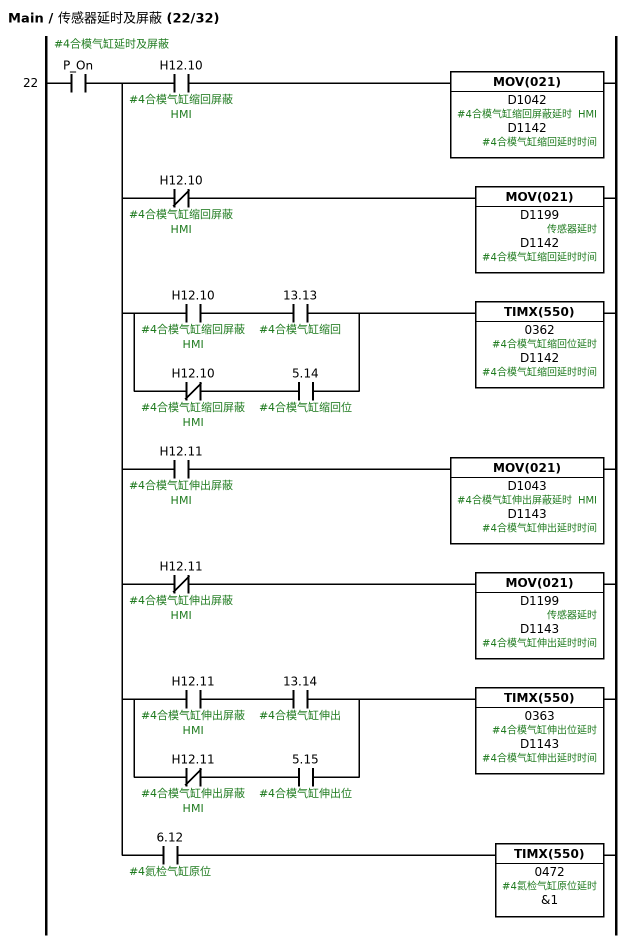
; [picture p24: Main / 传感器延时及屏蔽, rungs 22-22]
; rung 22: #4合模气缸延时及屏蔽
LD P_On
OUT TR0
AND H12.10  ; #4合模气缸缩回屏蔽  HMI
MOV(021) D1042 D1142  ; #4合模气缸缩回屏蔽延时  HMI, #4合模气缸缩回延时时间
LD TR0
ANDNOT H12.10  ; #4合模气缸缩回屏蔽  HMI
MOV(021) D1199 D1142  ; 传感器延时, #4合模气缸缩回延时时间
LD TR0
LD H12.10  ; #4合模气缸缩回屏蔽  HMI
AND 13.13  ; #4合模气缸缩回
LDNOT H12.10  ; #4合模气缸缩回屏蔽  HMI
AND 5.14  ; #4合模气缸缩回位
ORLD
ANDLD
TIMX(550) 0362 D1142  ; #4合模气缸缩回延时时间, #4合模气缸缩回位延时
LD TR0
AND H12.11  ; #4合模气缸伸出屏蔽  HMI
MOV(021) D1043 D1143  ; #4合模气缸伸出屏蔽延时  HMI, #4合模气缸伸出延时时间
LD TR0
ANDNOT H12.11  ; #4合模气缸伸出屏蔽  HMI
MOV(021) D1199 D1143  ; 传感器延时, #4合模气缸伸出延时时间
LD TR0
LD H12.11  ; #4合模气缸伸出屏蔽  HMI
AND 13.14  ; #4合模气缸伸出
LDNOT H12.11  ; #4合模气缸伸出屏蔽  HMI
AND 5.15  ; #4合模气缸伸出位
ORLD
ANDLD
TIMX(550) 0363 D1143  ; #4合模气缸伸出延时时间, #4合模气缸伸出位延时
LD TR0
AND 6.12  ; #4氦检气缸原位
TIMX(550) 0472 &1  ; #4氦检气缸原位延时

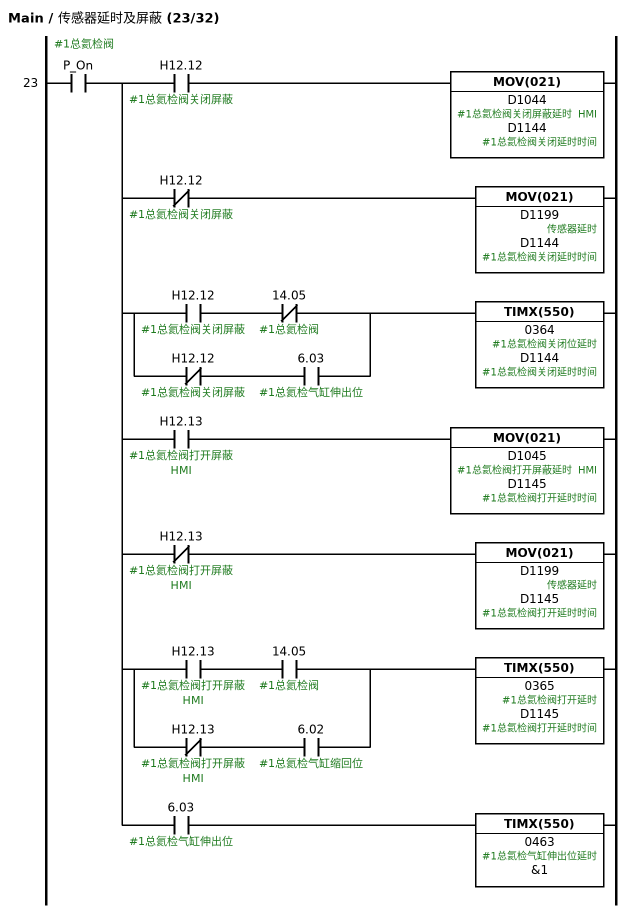
; rung 23: #1总氦检阀
LD P_On
OUT TR0
AND H12.12  ; #1总氦检阀关闭屏蔽
MOV(021) D1044 D1144  ; #1总氦检阀关闭屏蔽延时  HMI, #1总氦检阀关闭延时时间
LD TR0
ANDNOT H12.12  ; #1总氦检阀关闭屏蔽
MOV(021) D1199 D1144  ; 传感器延时, #1总氦检阀关闭延时时间
LD TR0
LD H12.12  ; #1总氦检阀关闭屏蔽
ANDNOT 14.05  ; #1总氦检阀
LDNOT H12.12  ; #1总氦检阀关闭屏蔽
AND 6.03  ; #1总氦检气缸伸出位
ORLD
ANDLD
TIMX(550) 0364 D1144  ; #1总氦检阀关闭延时时间, #1总氦检阀关闭位延时
LD TR0
AND H12.13  ; #1总氦检阀打开屏蔽  HMI
MOV(021) D1045 D1145  ; #1总氦检阀打开屏蔽延时  HMI, #1总氦检阀打开延时时间
LD TR0
ANDNOT H12.13  ; #1总氦检阀打开屏蔽  HMI
MOV(021) D1199 D1145  ; 传感器延时, #1总氦检阀打开延时时间
LD TR0
LD H12.13  ; #1总氦检阀打开屏蔽  HMI
AND 14.05  ; #1总氦检阀
LDNOT H12.13  ; #1总氦检阀打开屏蔽  HMI
AND 6.02  ; #1总氦检气缸缩回位
ORLD
ANDLD
TIMX(550) 0365 D1145  ; #1总氦检阀打开延时时间, #1总氦检阀打开延时
LD TR0
AND 6.03  ; #1总氦检气缸伸出位
TIMX(550) 0463 &1  ; #1总氦检气缸伸出位延时

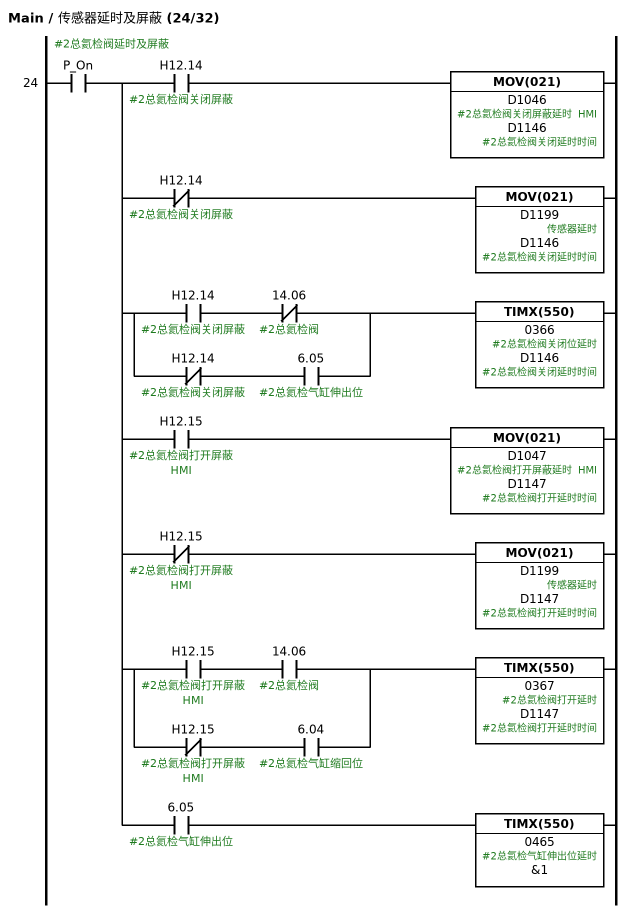
; rung 24: #2总氦检阀延时及屏蔽
LD P_On
OUT TR0
AND H12.14  ; #2总氦检阀关闭屏蔽
MOV(021) D1046 D1146  ; #2总氦检阀关闭屏蔽延时  HMI, #2总氦检阀关闭延时时间
LD TR0
ANDNOT H12.14  ; #2总氦检阀关闭屏蔽
MOV(021) D1199 D1146  ; 传感器延时, #2总氦检阀关闭延时时间
LD TR0
LD H12.14  ; #2总氦检阀关闭屏蔽
ANDNOT 14.06  ; #2总氦检阀
LDNOT H12.14  ; #2总氦检阀关闭屏蔽
AND 6.05  ; #2总氦检气缸伸出位
ORLD
ANDLD
TIMX(550) 0366 D1146  ; #2总氦检阀关闭延时时间, #2总氦检阀关闭位延时
LD TR0
AND H12.15  ; #2总氦检阀打开屏蔽  HMI
MOV(021) D1047 D1147  ; #2总氦检阀打开屏蔽延时  HMI, #2总氦检阀打开延时时间
LD TR0
ANDNOT H12.15  ; #2总氦检阀打开屏蔽  HMI
MOV(021) D1199 D1147  ; 传感器延时, #2总氦检阀打开延时时间
LD TR0
LD H12.15  ; #2总氦检阀打开屏蔽  HMI
AND 14.06  ; #2总氦检阀
LDNOT H12.15  ; #2总氦检阀打开屏蔽  HMI
AND 6.04  ; #2总氦检气缸缩回位
ORLD
ANDLD
TIMX(550) 0367 D1147  ; #2总氦检阀打开延时时间, #2总氦检阀打开延时
LD TR0
AND 6.05  ; #2总氦检气缸伸出位
TIMX(550) 0465 &1  ; #2总氦检气缸伸出位延时

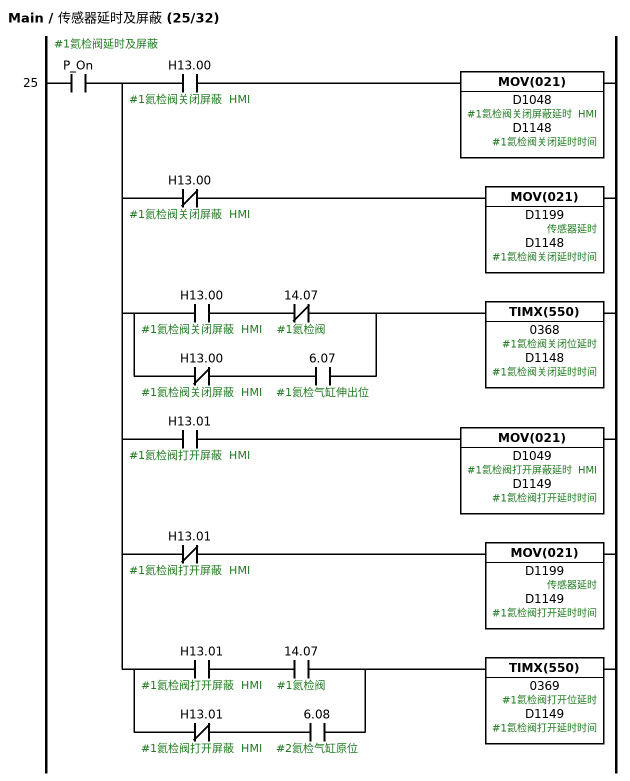
; rung 25: #1氦检阀延时及屏蔽
LD P_On
OUT TR0
AND H13.00  ; #1氦检阀关闭屏蔽  HMI
MOV(021) D1048 D1148  ; #1氦检阀关闭屏蔽延时  HMI, #1氦检阀关闭延时时间
LD TR0
ANDNOT H13.00  ; #1氦检阀关闭屏蔽  HMI
MOV(021) D1199 D1148  ; 传感器延时, #1氦检阀关闭延时时间
LD TR0
LD H13.00  ; #1氦检阀关闭屏蔽  HMI
ANDNOT 14.07  ; #1氦检阀
LDNOT H13.00  ; #1氦检阀关闭屏蔽  HMI
AND 6.07  ; #1氦检气缸伸出位
ORLD
ANDLD
TIMX(550) 0368 D1148  ; #1氦检阀关闭延时时间, #1氦检阀关闭位延时
LD TR0
AND H13.01  ; #1氦检阀打开屏蔽  HMI
MOV(021) D1049 D1149  ; #1氦检阀打开屏蔽延时  HMI, #1氦检阀打开延时时间
LD TR0
ANDNOT H13.01  ; #1氦检阀打开屏蔽  HMI
MOV(021) D1199 D1149  ; 传感器延时, #1氦检阀打开延时时间
LD TR0
LD H13.01  ; #1氦检阀打开屏蔽  HMI
AND 14.07  ; #1氦检阀
LDNOT H13.01  ; #1氦检阀打开屏蔽  HMI
AND 6.08  ; #2氦检气缸原位
ORLD
ANDLD
TIMX(550) 0369 D1149  ; #1氦检阀打开延时时间, #1氦检阀打开位延时

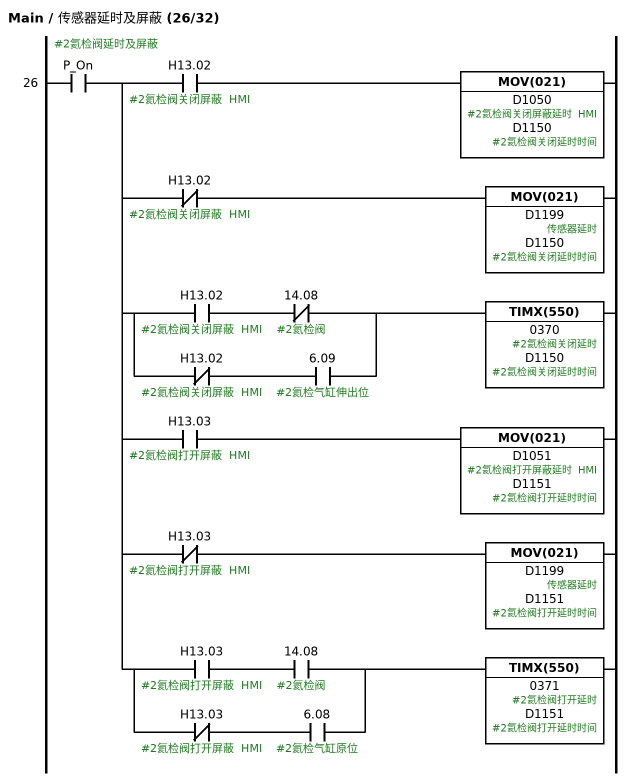
; rung 26: #2氦检阀延时及屏蔽
LD P_On
OUT TR0
AND H13.02  ; #2氦检阀关闭屏蔽  HMI
MOV(021) D1050 D1150  ; #2氦检阀关闭屏蔽延时  HMI, #2氦检阀关闭延时时间
LD TR0
ANDNOT H13.02  ; #2氦检阀关闭屏蔽  HMI
MOV(021) D1199 D1150  ; 传感器延时, #2氦检阀关闭延时时间
LD TR0
LD H13.02  ; #2氦检阀关闭屏蔽  HMI
ANDNOT 14.08  ; #2氦检阀
LDNOT H13.02  ; #2氦检阀关闭屏蔽  HMI
AND 6.09  ; #2氦检气缸伸出位
ORLD
ANDLD
TIMX(550) 0370 D1150  ; #2氦检阀关闭延时时间, #2氦检阀关闭延时
LD TR0
AND H13.03  ; #2氦检阀打开屏蔽  HMI
MOV(021) D1051 D1151  ; #2氦检阀打开屏蔽延时  HMI, #2氦检阀打开延时时间
LD TR0
ANDNOT H13.03  ; #2氦检阀打开屏蔽  HMI
MOV(021) D1199 D1151  ; 传感器延时, #2氦检阀打开延时时间
LD TR0
LD H13.03  ; #2氦检阀打开屏蔽  HMI
AND 14.08  ; #2氦检阀
LDNOT H13.03  ; #2氦检阀打开屏蔽  HMI
AND 6.08  ; #2氦检气缸原位
ORLD
ANDLD
TIMX(550) 0371 D1151  ; #2氦检阀打开延时时间, #2氦检阀打开延时

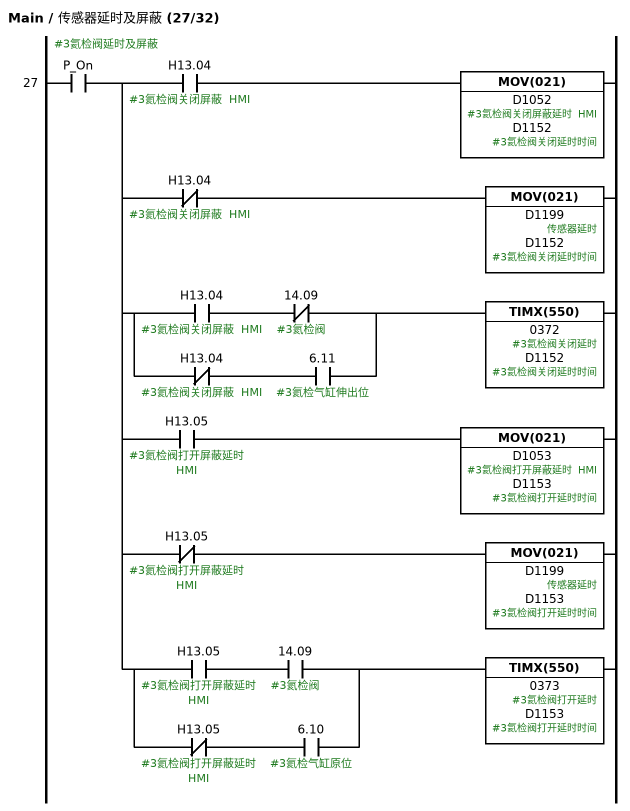
; rung 27: #3氦检阀延时及屏蔽
LD P_On
OUT TR0
AND H13.04  ; #3氦检阀关闭屏蔽  HMI
MOV(021) D1052 D1152  ; #3氦检阀关闭屏蔽延时  HMI, #3氦检阀关闭延时时间
LD TR0
ANDNOT H13.04  ; #3氦检阀关闭屏蔽  HMI
MOV(021) D1199 D1152  ; 传感器延时, #3氦检阀关闭延时时间
LD TR0
LD H13.04  ; #3氦检阀关闭屏蔽  HMI
ANDNOT 14.09  ; #3氦检阀
LDNOT H13.04  ; #3氦检阀关闭屏蔽  HMI
AND 6.11  ; #3氦检气缸伸出位
ORLD
ANDLD
TIMX(550) 0372 D1152  ; #3氦检阀关闭延时时间, #3氦检阀关闭延时
LD TR0
AND H13.05  ; #3氦检阀打开屏蔽延时  HMI
MOV(021) D1053 D1153  ; #3氦检阀打开屏蔽延时  HMI, #3氦检阀打开延时时间
LD TR0
ANDNOT H13.05  ; #3氦检阀打开屏蔽延时  HMI
MOV(021) D1199 D1153  ; 传感器延时, #3氦检阀打开延时时间
LD TR0
LD H13.05  ; #3氦检阀打开屏蔽延时  HMI
AND 14.09  ; #3氦检阀
LDNOT H13.05  ; #3氦检阀打开屏蔽延时  HMI
AND 6.10  ; #3氦检气缸原位
ORLD
ANDLD
TIMX(550) 0373 D1153  ; #3氦检阀打开延时时间, #3氦检阀打开延时

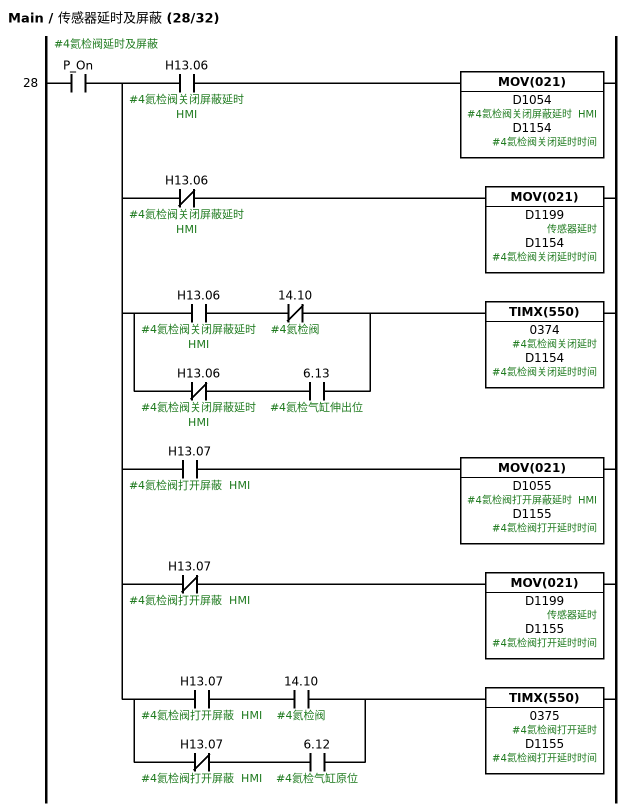
; rung 28: #4氦检阀延时及屏蔽
LD P_On
OUT TR0
AND H13.06  ; #4氦检阀关闭屏蔽延时  HMI
MOV(021) D1054 D1154  ; #4氦检阀关闭屏蔽延时  HMI, #4氦检阀关闭延时时间
LD TR0
ANDNOT H13.06  ; #4氦检阀关闭屏蔽延时  HMI
MOV(021) D1199 D1154  ; 传感器延时, #4氦检阀关闭延时时间
LD TR0
LD H13.06  ; #4氦检阀关闭屏蔽延时  HMI
ANDNOT 14.10  ; #4氦检阀
LDNOT H13.06  ; #4氦检阀关闭屏蔽延时  HMI
AND 6.13  ; #4氦检气缸伸出位
ORLD
ANDLD
TIMX(550) 0374 D1154  ; #4氦检阀关闭延时时间, #4氦检阀关闭延时
LD TR0
AND H13.07  ; #4氦检阀打开屏蔽  HMI
MOV(021) D1055 D1155  ; #4氦检阀打开屏蔽延时  HMI, #4氦检阀打开延时时间
LD TR0
ANDNOT H13.07  ; #4氦检阀打开屏蔽  HMI
MOV(021) D1199 D1155  ; 传感器延时, #4氦检阀打开延时时间
LD TR0
LD H13.07  ; #4氦检阀打开屏蔽  HMI
AND 14.10  ; #4氦检阀
LDNOT H13.07  ; #4氦检阀打开屏蔽  HMI
AND 6.12  ; #4氦检气缸原位
ORLD
ANDLD
TIMX(550) 0375 D1155  ; #4氦检阀打开延时时间, #4氦检阀打开延时

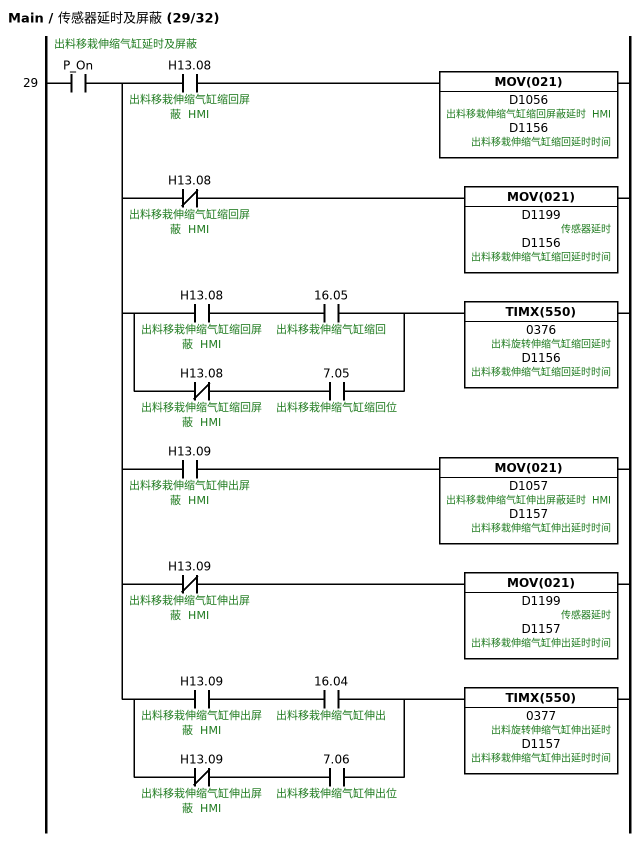
; rung 29: 出料移栽伸缩气缸延时及屏蔽
LD P_On
OUT TR0
AND H13.08  ; 出料移栽伸缩气缸缩回屏蔽  HMI
MOV(021) D1056 D1156  ; 出料移栽伸缩气缸缩回屏蔽延时  HMI, 出料移栽伸缩气缸缩回延时时间
LD TR0
ANDNOT H13.08  ; 出料移栽伸缩气缸缩回屏蔽  HMI
MOV(021) D1199 D1156  ; 传感器延时, 出料移栽伸缩气缸缩回延时时间
LD TR0
LD H13.08  ; 出料移栽伸缩气缸缩回屏蔽  HMI
AND 16.05  ; 出料移栽伸缩气缸缩回
LDNOT H13.08  ; 出料移栽伸缩气缸缩回屏蔽  HMI
AND 7.05  ; 出料移栽伸缩气缸缩回位
ORLD
ANDLD
TIMX(550) 0376 D1156  ; 出料移栽伸缩气缸缩回延时时间, 出料旋转伸缩气缸缩回延时
LD TR0
AND H13.09  ; 出料移栽伸缩气缸伸出屏蔽  HMI
MOV(021) D1057 D1157  ; 出料移栽伸缩气缸伸出屏蔽延时  HMI, 出料移栽伸缩气缸伸出延时时间
LD TR0
ANDNOT H13.09  ; 出料移栽伸缩气缸伸出屏蔽  HMI
MOV(021) D1199 D1157  ; 传感器延时, 出料移栽伸缩气缸伸出延时时间
LD TR0
LD H13.09  ; 出料移栽伸缩气缸伸出屏蔽  HMI
AND 16.04  ; 出料移栽伸缩气缸伸出
LDNOT H13.09  ; 出料移栽伸缩气缸伸出屏蔽  HMI
AND 7.06  ; 出料移栽伸缩气缸伸出位
ORLD
ANDLD
TIMX(550) 0377 D1157  ; 出料移栽伸缩气缸伸出延时时间, 出料旋转伸缩气缸伸出延时

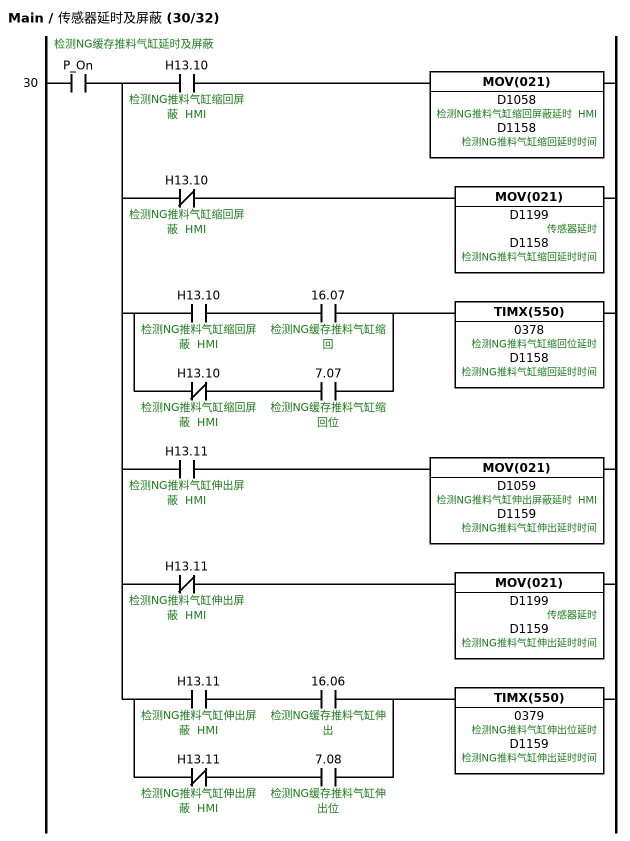
; rung 30: 检测NG缓存推料气缸延时及屏蔽
LD P_On
OUT TR0
AND H13.10  ; 检测NG推料气缸缩回屏蔽  HMI
MOV(021) D1058 D1158  ; 检测NG推料气缸缩回屏蔽延时  HMI, 检测NG推料气缸缩回延时时间
LD TR0
ANDNOT H13.10  ; 检测NG推料气缸缩回屏蔽  HMI
MOV(021) D1199 D1158  ; 传感器延时, 检测NG推料气缸缩回延时时间
LD TR0
LD H13.10  ; 检测NG推料气缸缩回屏蔽  HMI
AND 16.07  ; 检测NG缓存推料气缸缩回
LDNOT H13.10  ; 检测NG推料气缸缩回屏蔽  HMI
AND 7.07  ; 检测NG缓存推料气缸缩回位
ORLD
ANDLD
TIMX(550) 0378 D1158  ; 检测NG推料气缸缩回延时时间, 检测NG推料气缸缩回位延时
LD TR0
AND H13.11  ; 检测NG推料气缸伸出屏蔽  HMI
MOV(021) D1059 D1159  ; 检测NG推料气缸伸出屏蔽延时  HMI, 检测NG推料气缸伸出延时时间
LD TR0
ANDNOT H13.11  ; 检测NG推料气缸伸出屏蔽  HMI
MOV(021) D1199 D1159  ; 传感器延时, 检测NG推料气缸伸出延时时间
LD TR0
LD H13.11  ; 检测NG推料气缸伸出屏蔽  HMI
AND 16.06  ; 检测NG缓存推料气缸伸出
LDNOT H13.11  ; 检测NG推料气缸伸出屏蔽  HMI
AND 7.08  ; 检测NG缓存推料气缸伸出位
ORLD
ANDLD
TIMX(550) 0379 D1159  ; 检测NG推料气缸伸出延时时间, 检测NG推料气缸伸出位延时

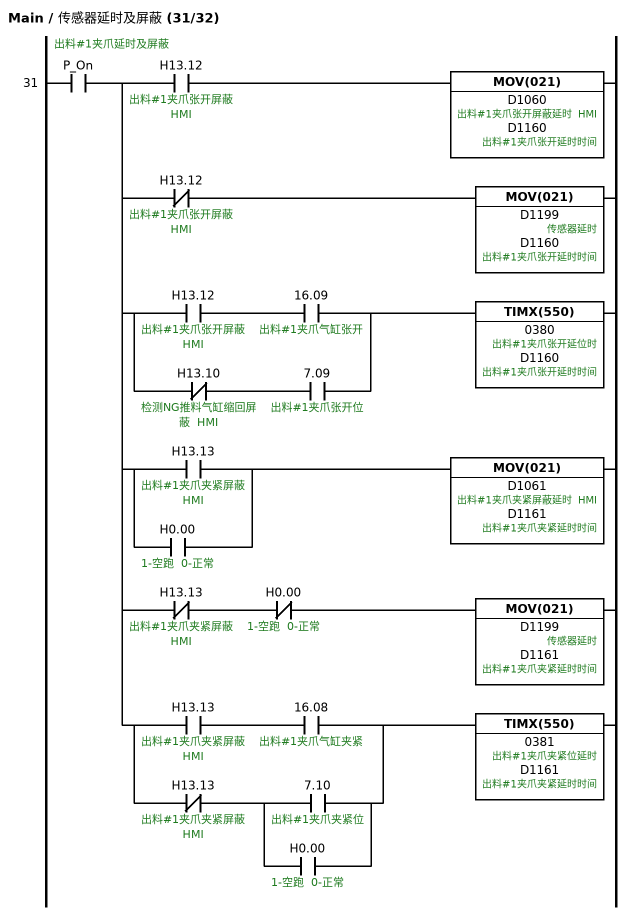
; rung 31: 出料#1夹爪延时及屏蔽
LD P_On
OUT TR0
AND H13.12  ; 出料#1夹爪张开屏蔽  HMI
MOV(021) D1060 D1160  ; 出料#1夹爪张开屏蔽延时  HMI, 出料#1夹爪张开延时时间
LD TR0
ANDNOT H13.12  ; 出料#1夹爪张开屏蔽  HMI
MOV(021) D1199 D1160  ; 传感器延时, 出料#1夹爪张开延时时间
LD TR0
LD H13.12  ; 出料#1夹爪张开屏蔽  HMI
AND 16.09  ; 出料#1夹爪气缸张开
LDNOT H13.10  ; 检测NG推料气缸缩回屏蔽  HMI
AND 7.09  ; 出料#1夹爪张开位
ORLD
ANDLD
TIMX(550) 0380 D1160  ; 出料#1夹爪张开延时时间, 出料#1夹爪张开延位时
LD TR0
LD H13.13  ; 出料#1夹爪夹紧屏蔽  HMI
OR H0.00  ; 1-空跑  0-正常
ANDLD
MOV(021) D1061 D1161  ; 出料#1夹爪夹紧屏蔽延时  HMI, 出料#1夹爪夹紧延时时间
LD TR0
ANDNOT H13.13  ; 出料#1夹爪夹紧屏蔽  HMI
ANDNOT H0.00  ; 1-空跑  0-正常
MOV(021) D1199 D1161  ; 传感器延时, 出料#1夹爪夹紧延时时间
LD TR0
LD H13.13  ; 出料#1夹爪夹紧屏蔽  HMI
AND 16.08  ; 出料#1夹爪气缸夹紧
LDNOT H13.13  ; 出料#1夹爪夹紧屏蔽  HMI
LD 7.10  ; 出料#1夹爪夹紧位
OR H0.00  ; 1-空跑  0-正常
ANDLD
ORLD
ANDLD
TIMX(550) 0381 D1161  ; 出料#1夹爪夹紧延时时间, 出料#1夹爪夹紧位延时

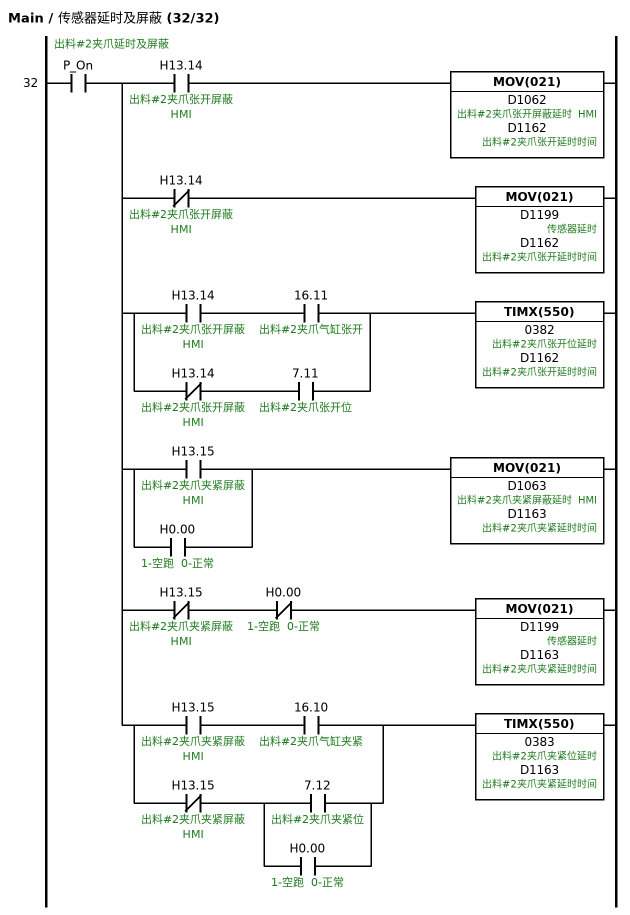
; rung 32: 出料#2夹爪延时及屏蔽
LD P_On
OUT TR0
AND H13.14  ; 出料#2夹爪张开屏蔽  HMI
MOV(021) D1062 D1162  ; 出料#2夹爪张开屏蔽延时  HMI, 出料#2夹爪张开延时时间
LD TR0
ANDNOT H13.14  ; 出料#2夹爪张开屏蔽  HMI
MOV(021) D1199 D1162  ; 传感器延时, 出料#2夹爪张开延时时间
LD TR0
LD H13.14  ; 出料#2夹爪张开屏蔽  HMI
AND 16.11  ; 出料#2夹爪气缸张开
LDNOT H13.14  ; 出料#2夹爪张开屏蔽  HMI
AND 7.11  ; 出料#2夹爪张开位
ORLD
ANDLD
TIMX(550) 0382 D1162  ; 出料#2夹爪张开延时时间, 出料#2夹爪张开位延时
LD TR0
LD H13.15  ; 出料#2夹爪夹紧屏蔽  HMI
OR H0.00  ; 1-空跑  0-正常
ANDLD
MOV(021) D1063 D1163  ; 出料#2夹爪夹紧屏蔽延时  HMI, 出料#2夹爪夹紧延时时间
LD TR0
ANDNOT H13.15  ; 出料#2夹爪夹紧屏蔽  HMI
ANDNOT H0.00  ; 1-空跑  0-正常
MOV(021) D1199 D1163  ; 传感器延时, 出料#2夹爪夹紧延时时间
LD TR0
LD H13.15  ; 出料#2夹爪夹紧屏蔽  HMI
AND 16.10  ; 出料#2夹爪气缸夹紧
LDNOT H13.15  ; 出料#2夹爪夹紧屏蔽  HMI
LD 7.12  ; 出料#2夹爪夹紧位
OR H0.00  ; 1-空跑  0-正常
ANDLD
ORLD
ANDLD
TIMX(550) 0383 D1163  ; 出料#2夹爪夹紧延时时间, 出料#2夹爪夹紧位延时

### Section 报警

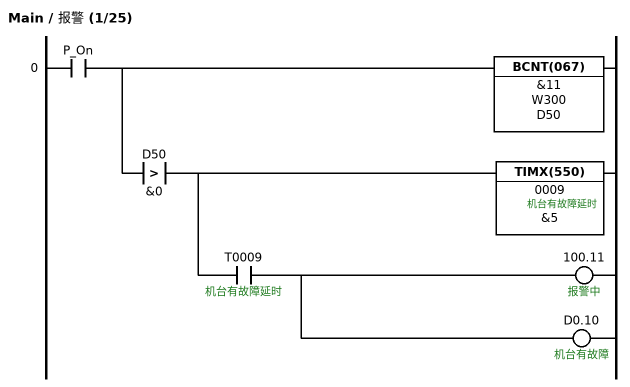
; rung 0
LD P_On
BCNT(067) &11 W300 D50
AND>(320) D50 &0
TIMX(550) 0009 &5  ; 机台有故障延时
AND T0009  ; 机台有故障延时
OUT 100.11  ; 报警中
OUT D0.10  ; 机台有故障

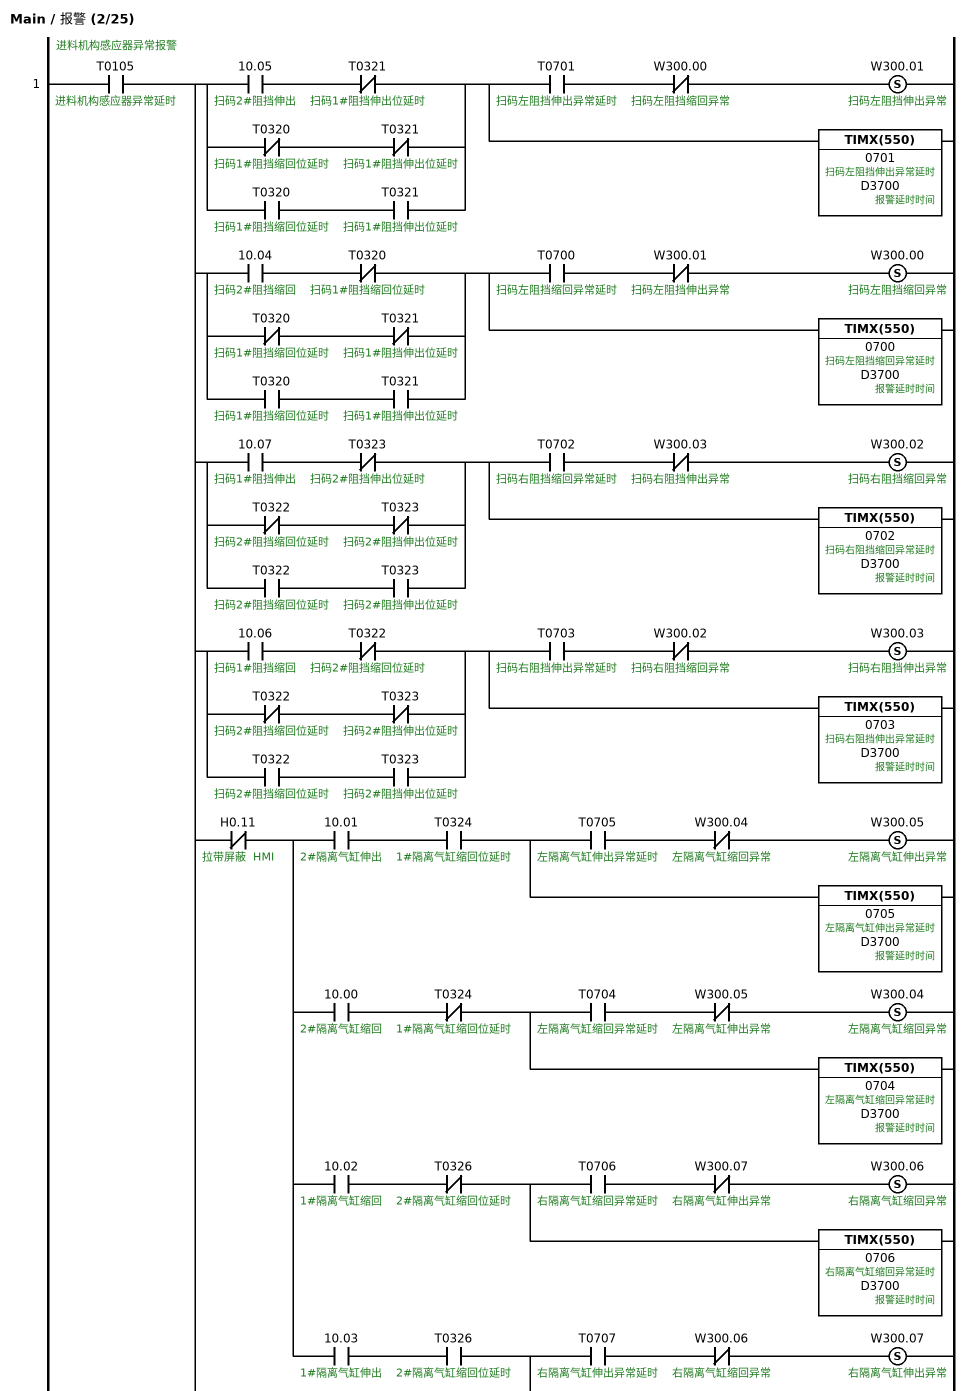

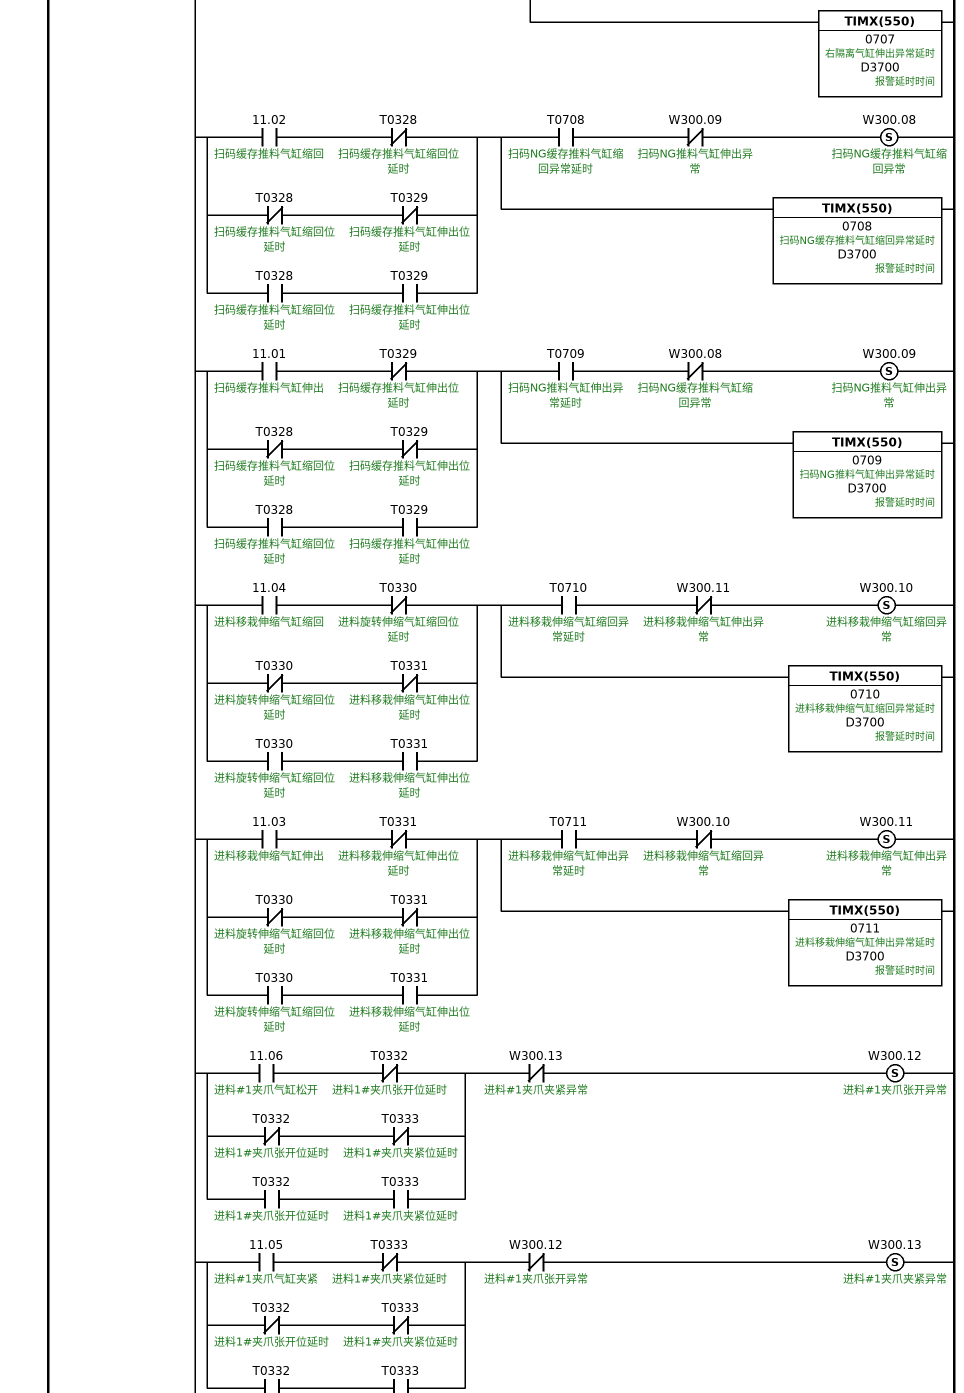

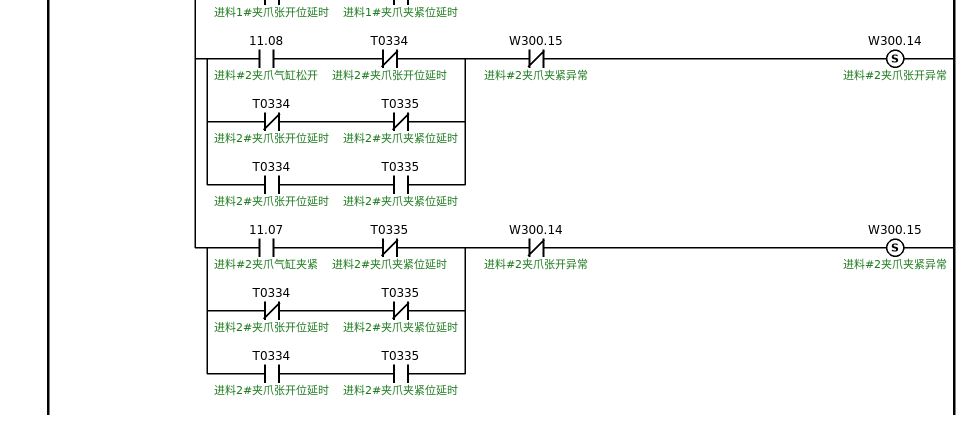
; rung 1: 进料机构感应器异常报警
LD T0105  ; 进料机构感应器异常延时
OUT TR0
LD 10.05  ; 扫码2#阻挡伸出
ANDNOT T0321  ; 扫码1#阻挡伸出位延时
LDNOT T0320  ; 扫码1#阻挡缩回位延时
ANDNOT T0321  ; 扫码1#阻挡伸出位延时
ORLD
LD T0320  ; 扫码1#阻挡缩回位延时
AND T0321  ; 扫码1#阻挡伸出位延时
ORLD
ANDLD
OUT TR1
AND T0701  ; 扫码左阻挡伸出异常延时
ANDNOT W300.00  ; 扫码左阻挡缩回异常
SET W300.01  ; 扫码左阻挡伸出异常
LD TR1
TIMX(550) 0701 D3700  ; 报警延时时间, 扫码左阻挡伸出异常延时
LD TR0
LD 10.04  ; 扫码2#阻挡缩回
ANDNOT T0320  ; 扫码1#阻挡缩回位延时
LDNOT T0320  ; 扫码1#阻挡缩回位延时
ANDNOT T0321  ; 扫码1#阻挡伸出位延时
ORLD
LD T0320  ; 扫码1#阻挡缩回位延时
AND T0321  ; 扫码1#阻挡伸出位延时
ORLD
ANDLD
OUT TR1
AND T0700  ; 扫码左阻挡缩回异常延时
ANDNOT W300.01  ; 扫码左阻挡伸出异常
SET W300.00  ; 扫码左阻挡缩回异常
LD TR1
TIMX(550) 0700 D3700  ; 报警延时时间, 扫码左阻挡缩回异常延时
LD TR0
LD 10.07  ; 扫码1#阻挡伸出
ANDNOT T0323  ; 扫码2#阻挡伸出位延时
LDNOT T0322  ; 扫码2#阻挡缩回位延时
ANDNOT T0323  ; 扫码2#阻挡伸出位延时
ORLD
LD T0322  ; 扫码2#阻挡缩回位延时
AND T0323  ; 扫码2#阻挡伸出位延时
ORLD
ANDLD
OUT TR1
AND T0702  ; 扫码右阻挡缩回异常延时
ANDNOT W300.03  ; 扫码右阻挡伸出异常
SET W300.02  ; 扫码右阻挡缩回异常
LD TR1
TIMX(550) 0702 D3700  ; 报警延时时间, 扫码右阻挡缩回异常延时
LD TR0
LD 10.06  ; 扫码1#阻挡缩回
ANDNOT T0322  ; 扫码2#阻挡缩回位延时
LDNOT T0322  ; 扫码2#阻挡缩回位延时
ANDNOT T0323  ; 扫码2#阻挡伸出位延时
ORLD
LD T0322  ; 扫码2#阻挡缩回位延时
AND T0323  ; 扫码2#阻挡伸出位延时
ORLD
ANDLD
OUT TR1
AND T0703  ; 扫码右阻挡伸出异常延时
ANDNOT W300.02  ; 扫码右阻挡缩回异常
SET W300.03  ; 扫码右阻挡伸出异常
LD TR1
TIMX(550) 0703 D3700  ; 报警延时时间, 扫码右阻挡伸出异常延时
LD TR0
ANDNOT H0.11  ; 拉带屏蔽  HMI
OUT TR1
AND 10.01  ; 2#隔离气缸伸出
AND T0324  ; 1#隔离气缸缩回位延时
OUT TR2
AND T0705  ; 左隔离气缸伸出异常延时
ANDNOT W300.04  ; 左隔离气缸缩回异常
SET W300.05  ; 左隔离气缸伸出异常
LD TR2
TIMX(550) 0705 D3700  ; 报警延时时间, 左隔离气缸伸出异常延时
LD TR1
AND 10.00  ; 2#隔离气缸缩回
ANDNOT T0324  ; 1#隔离气缸缩回位延时
OUT TR2
AND T0704  ; 左隔离气缸缩回异常延时
ANDNOT W300.05  ; 左隔离气缸伸出异常
SET W300.04  ; 左隔离气缸缩回异常
LD TR2
TIMX(550) 0704 D3700  ; 报警延时时间, 左隔离气缸缩回异常延时
LD TR1
AND 10.02  ; 1#隔离气缸缩回
ANDNOT T0326  ; 2#隔离气缸缩回位延时
OUT TR2
AND T0706  ; 右隔离气缸缩回异常延时
ANDNOT W300.07  ; 右隔离气缸伸出异常
SET W300.06  ; 右隔离气缸缩回异常
LD TR2
TIMX(550) 0706 D3700  ; 报警延时时间, 右隔离气缸缩回异常延时
LD TR1
AND 10.03  ; 1#隔离气缸伸出
AND T0326  ; 2#隔离气缸缩回位延时
OUT TR1
AND T0707  ; 右隔离气缸伸出异常延时
ANDNOT W300.06  ; 右隔离气缸缩回异常
SET W300.07  ; 右隔离气缸伸出异常
LD TR1
TIMX(550) 0707 D3700  ; 报警延时时间, 右隔离气缸伸出异常延时
LD TR0
LD 11.02  ; 扫码缓存推料气缸缩回
ANDNOT T0328  ; 扫码缓存推料气缸缩回位延时
LDNOT T0328  ; 扫码缓存推料气缸缩回位延时
ANDNOT T0329  ; 扫码缓存推料气缸伸出位延时
ORLD
LD T0328  ; 扫码缓存推料气缸缩回位延时
AND T0329  ; 扫码缓存推料气缸伸出位延时
ORLD
ANDLD
OUT TR1
AND T0708  ; 扫码NG缓存推料气缸缩回异常延时
ANDNOT W300.09  ; 扫码NG推料气缸伸出异常
SET W300.08  ; 扫码NG缓存推料气缸缩回异常
LD TR1
TIMX(550) 0708 D3700  ; 报警延时时间, 扫码NG缓存推料气缸缩回异常延时
LD TR0
LD 11.01  ; 扫码缓存推料气缸伸出
ANDNOT T0329  ; 扫码缓存推料气缸伸出位延时
LDNOT T0328  ; 扫码缓存推料气缸缩回位延时
ANDNOT T0329  ; 扫码缓存推料气缸伸出位延时
ORLD
LD T0328  ; 扫码缓存推料气缸缩回位延时
AND T0329  ; 扫码缓存推料气缸伸出位延时
ORLD
ANDLD
OUT TR1
AND T0709  ; 扫码NG推料气缸伸出异常延时
ANDNOT W300.08  ; 扫码NG缓存推料气缸缩回异常
SET W300.09  ; 扫码NG推料气缸伸出异常
LD TR1
TIMX(550) 0709 D3700  ; 报警延时时间, 扫码NG推料气缸伸出异常延时
LD TR0
LD 11.04  ; 进料移栽伸缩气缸缩回
ANDNOT T0330  ; 进料旋转伸缩气缸缩回位延时
LDNOT T0330  ; 进料旋转伸缩气缸缩回位延时
ANDNOT T0331  ; 进料移栽伸缩气缸伸出位延时
ORLD
LD T0330  ; 进料旋转伸缩气缸缩回位延时
AND T0331  ; 进料移栽伸缩气缸伸出位延时
ORLD
ANDLD
OUT TR1
AND T0710  ; 进料移栽伸缩气缸缩回异常延时
ANDNOT W300.11  ; 进料移栽伸缩气缸伸出异常
SET W300.10  ; 进料移栽伸缩气缸缩回异常
LD TR1
TIMX(550) 0710 D3700  ; 报警延时时间, 进料移栽伸缩气缸缩回异常延时
LD TR0
LD 11.03  ; 进料移栽伸缩气缸伸出
ANDNOT T0331  ; 进料移栽伸缩气缸伸出位延时
LDNOT T0330  ; 进料旋转伸缩气缸缩回位延时
ANDNOT T0331  ; 进料移栽伸缩气缸伸出位延时
ORLD
LD T0330  ; 进料旋转伸缩气缸缩回位延时
AND T0331  ; 进料移栽伸缩气缸伸出位延时
ORLD
ANDLD
OUT TR1
AND T0711  ; 进料移栽伸缩气缸伸出异常延时
ANDNOT W300.10  ; 进料移栽伸缩气缸缩回异常
SET W300.11  ; 进料移栽伸缩气缸伸出异常
LD TR1
TIMX(550) 0711 D3700  ; 报警延时时间, 进料移栽伸缩气缸伸出异常延时
LD TR0
LD 11.06  ; 进料#1夹爪气缸松开
ANDNOT T0332  ; 进料1#夹爪张开位延时
LDNOT T0332  ; 进料1#夹爪张开位延时
ANDNOT T0333  ; 进料1#夹爪夹紧位延时
ORLD
LD T0332  ; 进料1#夹爪张开位延时
AND T0333  ; 进料1#夹爪夹紧位延时
ORLD
ANDLD
ANDNOT W300.13  ; 进料#1夹爪夹紧异常
SET W300.12  ; 进料#1夹爪张开异常
LD TR0
LD 11.05  ; 进料#1夹爪气缸夹紧
ANDNOT T0333  ; 进料1#夹爪夹紧位延时
LDNOT T0332  ; 进料1#夹爪张开位延时
ANDNOT T0333  ; 进料1#夹爪夹紧位延时
ORLD
LD T0332  ; 进料1#夹爪张开位延时
AND T0333  ; 进料1#夹爪夹紧位延时
ORLD
ANDLD
ANDNOT W300.12  ; 进料#1夹爪张开异常
SET W300.13  ; 进料#1夹爪夹紧异常
LD TR0
LD 11.08  ; 进料#2夹爪气缸松开
ANDNOT T0334  ; 进料2#夹爪张开位延时
LDNOT T0334  ; 进料2#夹爪张开位延时
ANDNOT T0335  ; 进料2#夹爪夹紧位延时
ORLD
LD T0334  ; 进料2#夹爪张开位延时
AND T0335  ; 进料2#夹爪夹紧位延时
ORLD
ANDLD
ANDNOT W300.15  ; 进料#2夹爪夹紧异常
SET W300.14  ; 进料#2夹爪张开异常
LD TR0
LD 11.07  ; 进料#2夹爪气缸夹紧
ANDNOT T0335  ; 进料2#夹爪夹紧位延时
LDNOT T0334  ; 进料2#夹爪张开位延时
ANDNOT T0335  ; 进料2#夹爪夹紧位延时
ORLD
LD T0334  ; 进料2#夹爪张开位延时
AND T0335  ; 进料2#夹爪夹紧位延时
ORLD
ANDLD
ANDNOT W300.14  ; 进料#2夹爪张开异常
SET W300.15  ; 进料#2夹爪夹紧异常

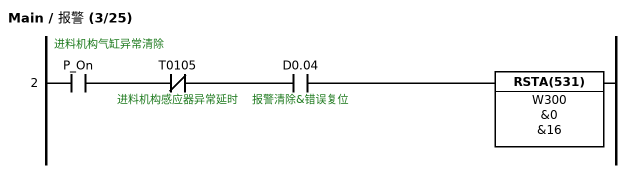
; rung 2: 进料机构气缸异常清除
LD P_On
ANDNOT T0105  ; 进料机构感应器异常延时
AND D0.04  ; 报警清除&错误复位
RSTA(531) W300 &0 &16

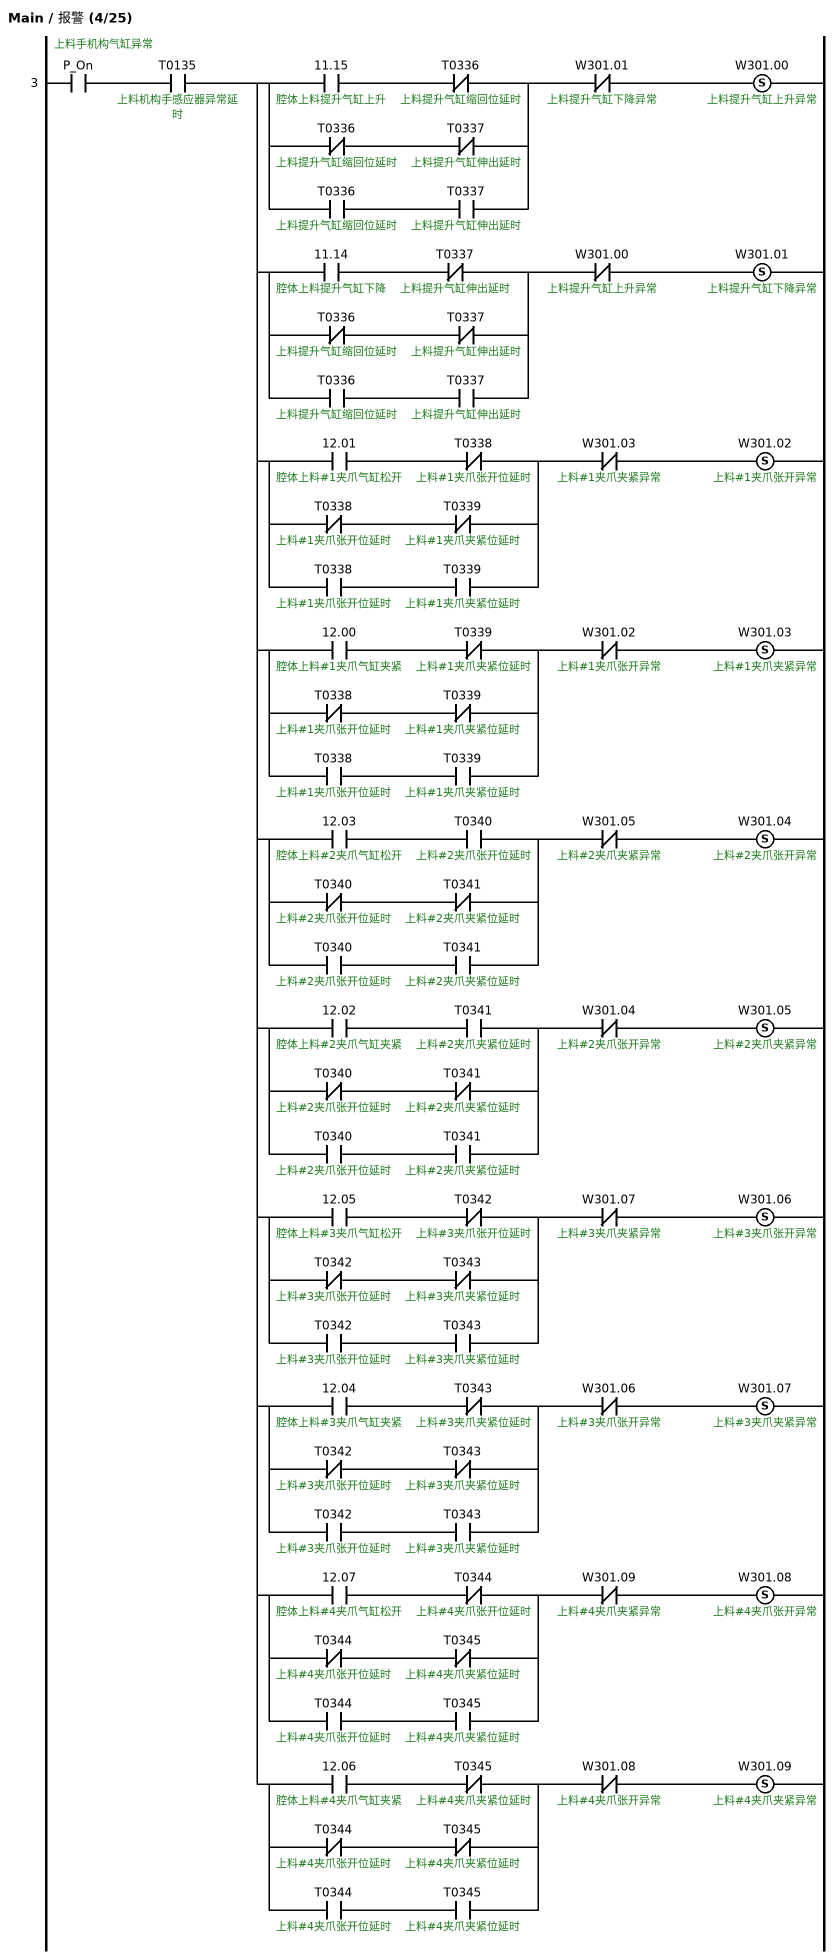
; rung 3: 上料手机构气缸异常
LD P_On
AND T0135  ; 上料机构手感应器异常延时
OUT TR0
LD 11.15  ; 腔体上料提升气缸上升
ANDNOT T0336  ; 上料提升气缸缩回位延时
LDNOT T0336  ; 上料提升气缸缩回位延时
ANDNOT T0337  ; 上料提升气缸伸出延时
ORLD
LD T0336  ; 上料提升气缸缩回位延时
AND T0337  ; 上料提升气缸伸出延时
ORLD
ANDLD
ANDNOT W301.01  ; 上料提升气缸下降异常
SET W301.00  ; 上料提升气缸上升异常
LD TR0
LD 11.14  ; 腔体上料提升气缸下降
ANDNOT T0337  ; 上料提升气缸伸出延时
LDNOT T0336  ; 上料提升气缸缩回位延时
ANDNOT T0337  ; 上料提升气缸伸出延时
ORLD
LD T0336  ; 上料提升气缸缩回位延时
AND T0337  ; 上料提升气缸伸出延时
ORLD
ANDLD
ANDNOT W301.00  ; 上料提升气缸上升异常
SET W301.01  ; 上料提升气缸下降异常
LD TR0
LD 12.01  ; 腔体上料#1夹爪气缸松开
ANDNOT T0338  ; 上料#1夹爪张开位延时
LDNOT T0338  ; 上料#1夹爪张开位延时
ANDNOT T0339  ; 上料#1夹爪夹紧位延时
ORLD
LD T0338  ; 上料#1夹爪张开位延时
AND T0339  ; 上料#1夹爪夹紧位延时
ORLD
ANDLD
ANDNOT W301.03  ; 上料#1夹爪夹紧异常
SET W301.02  ; 上料#1夹爪张开异常
LD TR0
LD 12.00  ; 腔体上料#1夹爪气缸夹紧
ANDNOT T0339  ; 上料#1夹爪夹紧位延时
LDNOT T0338  ; 上料#1夹爪张开位延时
ANDNOT T0339  ; 上料#1夹爪夹紧位延时
ORLD
LD T0338  ; 上料#1夹爪张开位延时
AND T0339  ; 上料#1夹爪夹紧位延时
ORLD
ANDLD
ANDNOT W301.02  ; 上料#1夹爪张开异常
SET W301.03  ; 上料#1夹爪夹紧异常
LD TR0
LD 12.03  ; 腔体上料#2夹爪气缸松开
AND T0340  ; 上料#2夹爪张开位延时
LDNOT T0340  ; 上料#2夹爪张开位延时
ANDNOT T0341  ; 上料#2夹爪夹紧位延时
ORLD
LD T0340  ; 上料#2夹爪张开位延时
AND T0341  ; 上料#2夹爪夹紧位延时
ORLD
ANDLD
ANDNOT W301.05  ; 上料#2夹爪夹紧异常
SET W301.04  ; 上料#2夹爪张开异常
LD TR0
LD 12.02  ; 腔体上料#2夹爪气缸夹紧
AND T0341  ; 上料#2夹爪夹紧位延时
LDNOT T0340  ; 上料#2夹爪张开位延时
ANDNOT T0341  ; 上料#2夹爪夹紧位延时
ORLD
LD T0340  ; 上料#2夹爪张开位延时
AND T0341  ; 上料#2夹爪夹紧位延时
ORLD
ANDLD
ANDNOT W301.04  ; 上料#2夹爪张开异常
SET W301.05  ; 上料#2夹爪夹紧异常
LD TR0
LD 12.05  ; 腔体上料#3夹爪气缸松开
ANDNOT T0342  ; 上料#3夹爪张开位延时
LDNOT T0342  ; 上料#3夹爪张开位延时
ANDNOT T0343  ; 上料#3夹爪夹紧位延时
ORLD
LD T0342  ; 上料#3夹爪张开位延时
AND T0343  ; 上料#3夹爪夹紧位延时
ORLD
ANDLD
ANDNOT W301.07  ; 上料#3夹爪夹紧异常
SET W301.06  ; 上料#3夹爪张开异常
LD TR0
LD 12.04  ; 腔体上料#3夹爪气缸夹紧
ANDNOT T0343  ; 上料#3夹爪夹紧位延时
LDNOT T0342  ; 上料#3夹爪张开位延时
ANDNOT T0343  ; 上料#3夹爪夹紧位延时
ORLD
LD T0342  ; 上料#3夹爪张开位延时
AND T0343  ; 上料#3夹爪夹紧位延时
ORLD
ANDLD
ANDNOT W301.06  ; 上料#3夹爪张开异常
SET W301.07  ; 上料#3夹爪夹紧异常
LD TR0
LD 12.07  ; 腔体上料#4夹爪气缸松开
ANDNOT T0344  ; 上料#4夹爪张开位延时
LDNOT T0344  ; 上料#4夹爪张开位延时
ANDNOT T0345  ; 上料#4夹爪夹紧位延时
ORLD
LD T0344  ; 上料#4夹爪张开位延时
AND T0345  ; 上料#4夹爪夹紧位延时
ORLD
ANDLD
ANDNOT W301.09  ; 上料#4夹爪夹紧异常
SET W301.08  ; 上料#4夹爪张开异常
LD TR0
LD 12.06  ; 腔体上料#4夹爪气缸夹紧
ANDNOT T0345  ; 上料#4夹爪夹紧位延时
LDNOT T0344  ; 上料#4夹爪张开位延时
ANDNOT T0345  ; 上料#4夹爪夹紧位延时
ORLD
LD T0344  ; 上料#4夹爪张开位延时
AND T0345  ; 上料#4夹爪夹紧位延时
ORLD
ANDLD
ANDNOT W301.08  ; 上料#4夹爪张开异常
SET W301.09  ; 上料#4夹爪夹紧异常

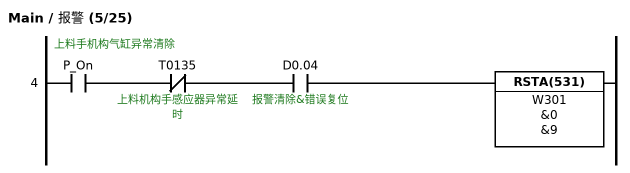
; rung 4: 上料手机构气缸异常清除
LD P_On
ANDNOT T0135  ; 上料机构手感应器异常延时
AND D0.04  ; 报警清除&错误复位
RSTA(531) W301 &0 &9

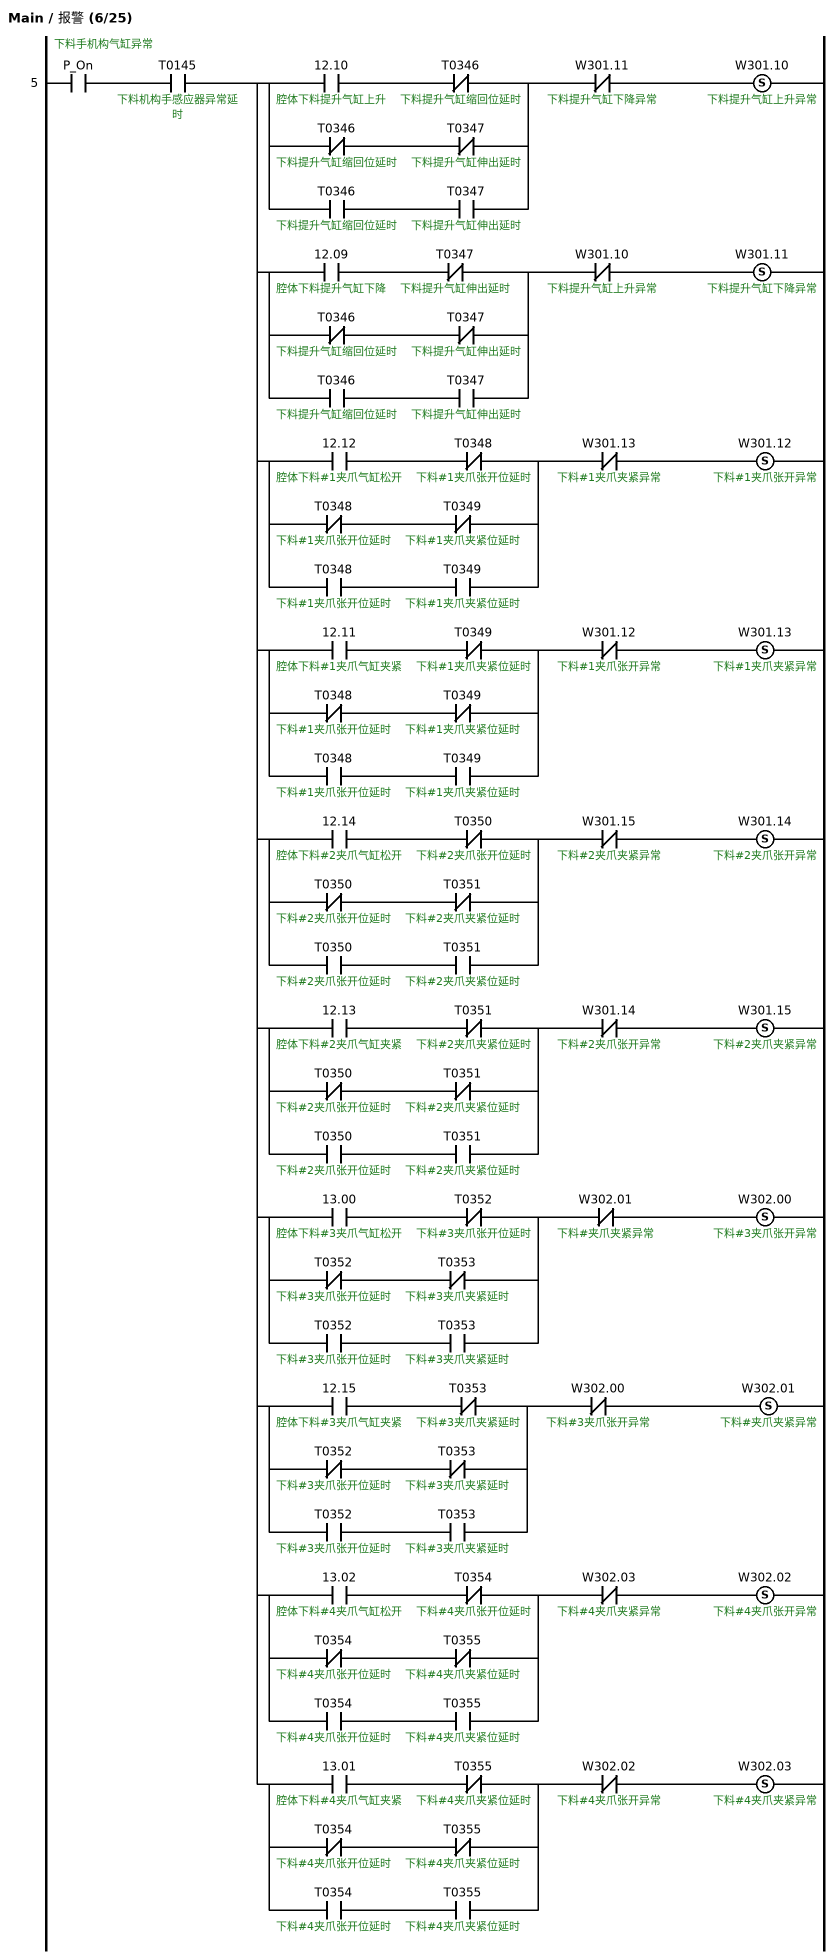
; rung 5: 下料手机构气缸异常
LD P_On
AND T0145  ; 下料机构手感应器异常延时
OUT TR0
LD 12.10  ; 腔体下料提升气缸上升
ANDNOT T0346  ; 下料提升气缸缩回位延时
LDNOT T0346  ; 下料提升气缸缩回位延时
ANDNOT T0347  ; 下料提升气缸伸出延时
ORLD
LD T0346  ; 下料提升气缸缩回位延时
AND T0347  ; 下料提升气缸伸出延时
ORLD
ANDLD
ANDNOT W301.11  ; 下料提升气缸下降异常
SET W301.10  ; 下料提升气缸上升异常
LD TR0
LD 12.09  ; 腔体下料提升气缸下降
ANDNOT T0347  ; 下料提升气缸伸出延时
LDNOT T0346  ; 下料提升气缸缩回位延时
ANDNOT T0347  ; 下料提升气缸伸出延时
ORLD
LD T0346  ; 下料提升气缸缩回位延时
AND T0347  ; 下料提升气缸伸出延时
ORLD
ANDLD
ANDNOT W301.10  ; 下料提升气缸上升异常
SET W301.11  ; 下料提升气缸下降异常
LD TR0
LD 12.12  ; 腔体下料#1夹爪气缸松开
ANDNOT T0348  ; 下料#1夹爪张开位延时
LDNOT T0348  ; 下料#1夹爪张开位延时
ANDNOT T0349  ; 下料#1夹爪夹紧位延时
ORLD
LD T0348  ; 下料#1夹爪张开位延时
AND T0349  ; 下料#1夹爪夹紧位延时
ORLD
ANDLD
ANDNOT W301.13  ; 下料#1夹爪夹紧异常
SET W301.12  ; 下料#1夹爪张开异常
LD TR0
LD 12.11  ; 腔体下料#1夹爪气缸夹紧
ANDNOT T0349  ; 下料#1夹爪夹紧位延时
LDNOT T0348  ; 下料#1夹爪张开位延时
ANDNOT T0349  ; 下料#1夹爪夹紧位延时
ORLD
LD T0348  ; 下料#1夹爪张开位延时
AND T0349  ; 下料#1夹爪夹紧位延时
ORLD
ANDLD
ANDNOT W301.12  ; 下料#1夹爪张开异常
SET W301.13  ; 下料#1夹爪夹紧异常
LD TR0
LD 12.14  ; 腔体下料#2夹爪气缸松开
ANDNOT T0350  ; 下料#2夹爪张开位延时
LDNOT T0350  ; 下料#2夹爪张开位延时
ANDNOT T0351  ; 下料#2夹爪夹紧位延时
ORLD
LD T0350  ; 下料#2夹爪张开位延时
AND T0351  ; 下料#2夹爪夹紧位延时
ORLD
ANDLD
ANDNOT W301.15  ; 下料#2夹爪夹紧异常
SET W301.14  ; 下料#2夹爪张开异常
LD TR0
LD 12.13  ; 腔体下料#2夹爪气缸夹紧
ANDNOT T0351  ; 下料#2夹爪夹紧位延时
LDNOT T0350  ; 下料#2夹爪张开位延时
ANDNOT T0351  ; 下料#2夹爪夹紧位延时
ORLD
LD T0350  ; 下料#2夹爪张开位延时
AND T0351  ; 下料#2夹爪夹紧位延时
ORLD
ANDLD
ANDNOT W301.14  ; 下料#2夹爪张开异常
SET W301.15  ; 下料#2夹爪夹紧异常
LD TR0
LD 13.00  ; 腔体下料#3夹爪气缸松开
ANDNOT T0352  ; 下料#3夹爪张开位延时
LDNOT T0352  ; 下料#3夹爪张开位延时
ANDNOT T0353  ; 下料#3夹爪夹紧延时
ORLD
LD T0352  ; 下料#3夹爪张开位延时
AND T0353  ; 下料#3夹爪夹紧延时
ORLD
ANDLD
ANDNOT W302.01  ; 下料#夹爪夹紧异常
SET W302.00  ; 下料#3夹爪张开异常
LD TR0
LD 12.15  ; 腔体下料#3夹爪气缸夹紧
ANDNOT T0353  ; 下料#3夹爪夹紧延时
LDNOT T0352  ; 下料#3夹爪张开位延时
ANDNOT T0353  ; 下料#3夹爪夹紧延时
ORLD
LD T0352  ; 下料#3夹爪张开位延时
AND T0353  ; 下料#3夹爪夹紧延时
ORLD
ANDLD
ANDNOT W302.00  ; 下料#3夹爪张开异常
SET W302.01  ; 下料#夹爪夹紧异常
LD TR0
LD 13.02  ; 腔体下料#4夹爪气缸松开
ANDNOT T0354  ; 下料#4夹爪张开位延时
LDNOT T0354  ; 下料#4夹爪张开位延时
ANDNOT T0355  ; 下料#4夹爪夹紧位延时
ORLD
LD T0354  ; 下料#4夹爪张开位延时
AND T0355  ; 下料#4夹爪夹紧位延时
ORLD
ANDLD
ANDNOT W302.03  ; 下料#4夹爪夹紧异常
SET W302.02  ; 下料#4夹爪张开异常
LD TR0
LD 13.01  ; 腔体下料#4夹爪气缸夹紧
ANDNOT T0355  ; 下料#4夹爪夹紧位延时
LDNOT T0354  ; 下料#4夹爪张开位延时
ANDNOT T0355  ; 下料#4夹爪夹紧位延时
ORLD
LD T0354  ; 下料#4夹爪张开位延时
AND T0355  ; 下料#4夹爪夹紧位延时
ORLD
ANDLD
ANDNOT W302.02  ; 下料#4夹爪张开异常
SET W302.03  ; 下料#4夹爪夹紧异常

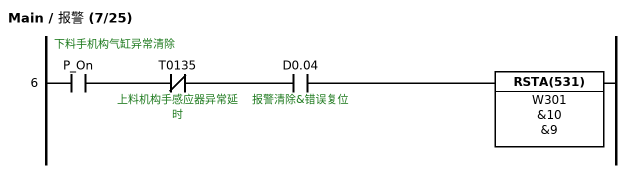
; rung 6: 下料手机构气缸异常清除
LD P_On
ANDNOT T0135  ; 上料机构手感应器异常延时
AND D0.04  ; 报警清除&错误复位
RSTA(531) W301 &10 &9

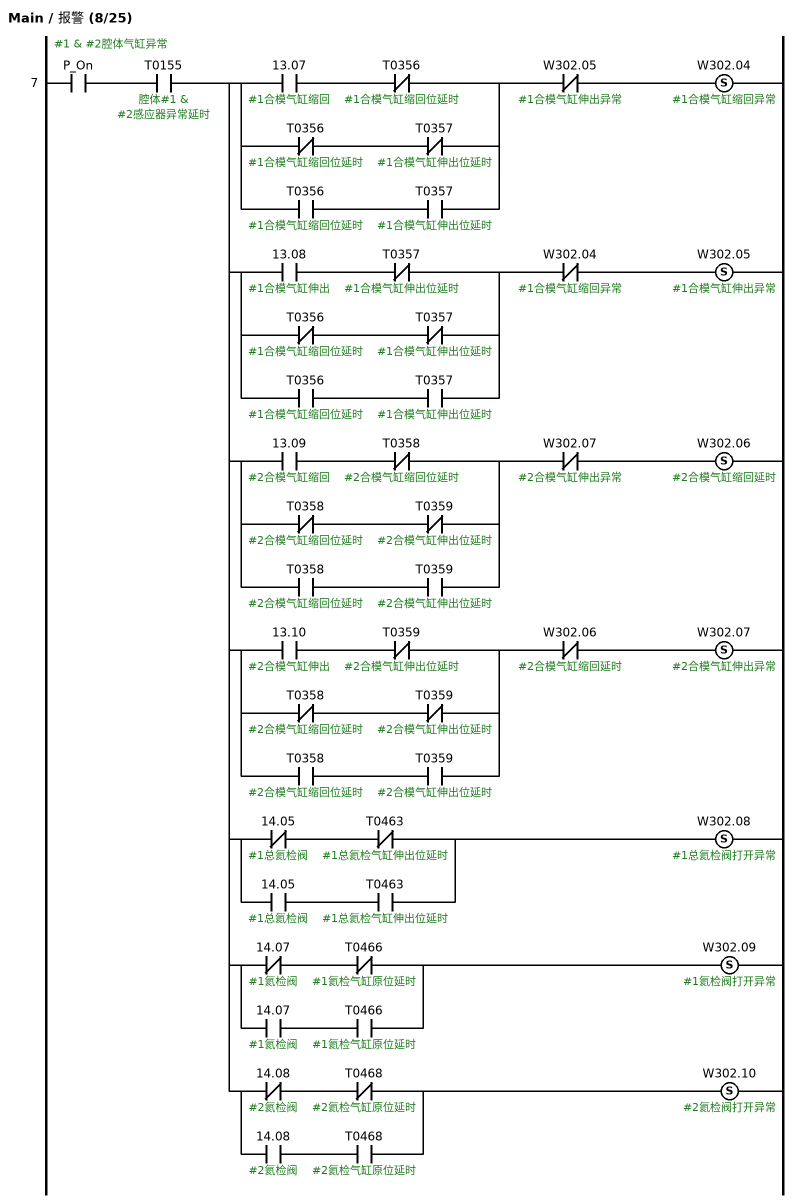
; rung 7: #1 & #2腔体气缸异常
LD P_On
AND T0155  ; 腔体#1 & #2感应器异常延时
OUT TR0
LD 13.07  ; #1合模气缸缩回
ANDNOT T0356  ; #1合模气缸缩回位延时
LDNOT T0356  ; #1合模气缸缩回位延时
ANDNOT T0357  ; #1合模气缸伸出位延时
ORLD
LD T0356  ; #1合模气缸缩回位延时
AND T0357  ; #1合模气缸伸出位延时
ORLD
ANDLD
ANDNOT W302.05  ; #1合模气缸伸出异常
SET W302.04  ; #1合模气缸缩回异常
LD TR0
LD 13.08  ; #1合模气缸伸出
ANDNOT T0357  ; #1合模气缸伸出位延时
LDNOT T0356  ; #1合模气缸缩回位延时
ANDNOT T0357  ; #1合模气缸伸出位延时
ORLD
LD T0356  ; #1合模气缸缩回位延时
AND T0357  ; #1合模气缸伸出位延时
ORLD
ANDLD
ANDNOT W302.04  ; #1合模气缸缩回异常
SET W302.05  ; #1合模气缸伸出异常
LD TR0
LD 13.09  ; #2合模气缸缩回
ANDNOT T0358  ; #2合模气缸缩回位延时
LDNOT T0358  ; #2合模气缸缩回位延时
ANDNOT T0359  ; #2合模气缸伸出位延时
ORLD
LD T0358  ; #2合模气缸缩回位延时
AND T0359  ; #2合模气缸伸出位延时
ORLD
ANDLD
ANDNOT W302.07  ; #2合模气缸伸出异常
SET W302.06  ; #2合模气缸缩回延时
LD TR0
LD 13.10  ; #2合模气缸伸出
ANDNOT T0359  ; #2合模气缸伸出位延时
LDNOT T0358  ; #2合模气缸缩回位延时
ANDNOT T0359  ; #2合模气缸伸出位延时
ORLD
LD T0358  ; #2合模气缸缩回位延时
AND T0359  ; #2合模气缸伸出位延时
ORLD
ANDLD
ANDNOT W302.06  ; #2合模气缸缩回延时
SET W302.07  ; #2合模气缸伸出异常
LD TR0
LDNOT 14.05  ; #1总氦检阀
ANDNOT T0463  ; #1总氦检气缸伸出位延时
LD 14.05  ; #1总氦检阀
AND T0463  ; #1总氦检气缸伸出位延时
ORLD
ANDLD
SET W302.08  ; #1总氦检阀打开异常
LD TR0
LDNOT 14.07  ; #1氦检阀
ANDNOT T0466  ; #1氦检气缸原位延时
LD 14.07  ; #1氦检阀
AND T0466  ; #1氦检气缸原位延时
ORLD
ANDLD
SET W302.09  ; #1氦检阀打开异常
LD TR0
LDNOT 14.08  ; #2氦检阀
ANDNOT T0468  ; #2氦检气缸原位延时
LD 14.08  ; #2氦检阀
AND T0468  ; #2氦检气缸原位延时
ORLD
ANDLD
SET W302.10  ; #2氦检阀打开异常

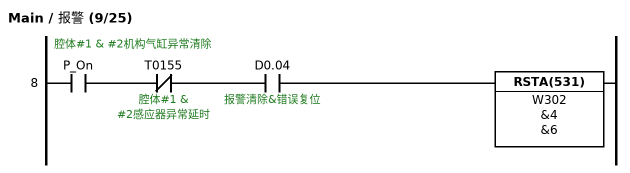
; rung 8: 腔体#1 & #2机构气缸异常清除
LD P_On
ANDNOT T0155  ; 腔体#1 & #2感应器异常延时
AND D0.04  ; 报警清除&错误复位
RSTA(531) W302 &4 &6

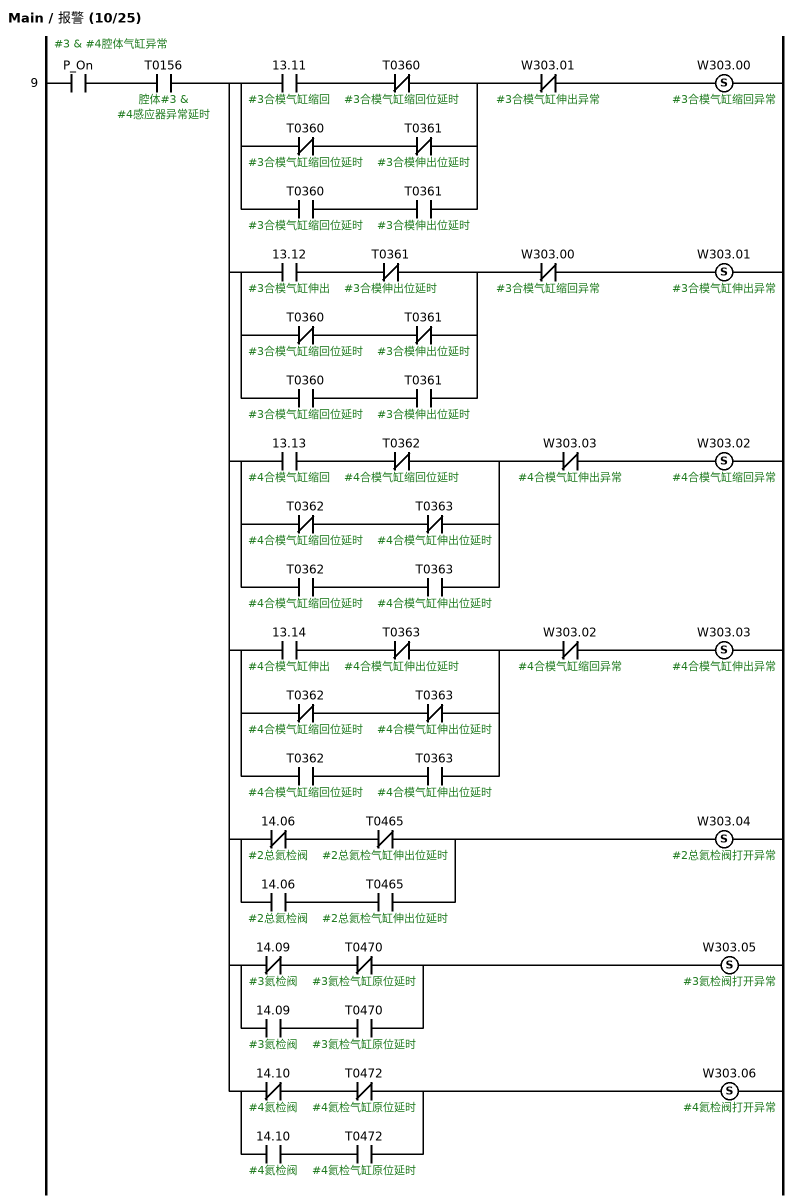
; rung 9: #3 & #4腔体气缸异常
LD P_On
AND T0156  ; 腔体#3 & #4感应器异常延时
OUT TR0
LD 13.11  ; #3合模气缸缩回
ANDNOT T0360  ; #3合模气缸缩回位延时
LDNOT T0360  ; #3合模气缸缩回位延时
ANDNOT T0361  ; #3合模伸出位延时
ORLD
LD T0360  ; #3合模气缸缩回位延时
AND T0361  ; #3合模伸出位延时
ORLD
ANDLD
ANDNOT W303.01  ; #3合模气缸伸出异常
SET W303.00  ; #3合模气缸缩回异常
LD TR0
LD 13.12  ; #3合模气缸伸出
ANDNOT T0361  ; #3合模伸出位延时
LDNOT T0360  ; #3合模气缸缩回位延时
ANDNOT T0361  ; #3合模伸出位延时
ORLD
LD T0360  ; #3合模气缸缩回位延时
AND T0361  ; #3合模伸出位延时
ORLD
ANDLD
ANDNOT W303.00  ; #3合模气缸缩回异常
SET W303.01  ; #3合模气缸伸出异常
LD TR0
LD 13.13  ; #4合模气缸缩回
ANDNOT T0362  ; #4合模气缸缩回位延时
LDNOT T0362  ; #4合模气缸缩回位延时
ANDNOT T0363  ; #4合模气缸伸出位延时
ORLD
LD T0362  ; #4合模气缸缩回位延时
AND T0363  ; #4合模气缸伸出位延时
ORLD
ANDLD
ANDNOT W303.03  ; #4合模气缸伸出异常
SET W303.02  ; #4合模气缸缩回异常
LD TR0
LD 13.14  ; #4合模气缸伸出
ANDNOT T0363  ; #4合模气缸伸出位延时
LDNOT T0362  ; #4合模气缸缩回位延时
ANDNOT T0363  ; #4合模气缸伸出位延时
ORLD
LD T0362  ; #4合模气缸缩回位延时
AND T0363  ; #4合模气缸伸出位延时
ORLD
ANDLD
ANDNOT W303.02  ; #4合模气缸缩回异常
SET W303.03  ; #4合模气缸伸出异常
LD TR0
LDNOT 14.06  ; #2总氦检阀
ANDNOT T0465  ; #2总氦检气缸伸出位延时
LD 14.06  ; #2总氦检阀
AND T0465  ; #2总氦检气缸伸出位延时
ORLD
ANDLD
SET W303.04  ; #2总氦检阀打开异常
LD TR0
LDNOT 14.09  ; #3氦检阀
ANDNOT T0470  ; #3氦检气缸原位延时
LD 14.09  ; #3氦检阀
AND T0470  ; #3氦检气缸原位延时
ORLD
ANDLD
SET W303.05  ; #3氦检阀打开异常
LD TR0
LDNOT 14.10  ; #4氦检阀
ANDNOT T0472  ; #4氦检气缸原位延时
LD 14.10  ; #4氦检阀
AND T0472  ; #4氦检气缸原位延时
ORLD
ANDLD
SET W303.06  ; #4氦检阀打开异常

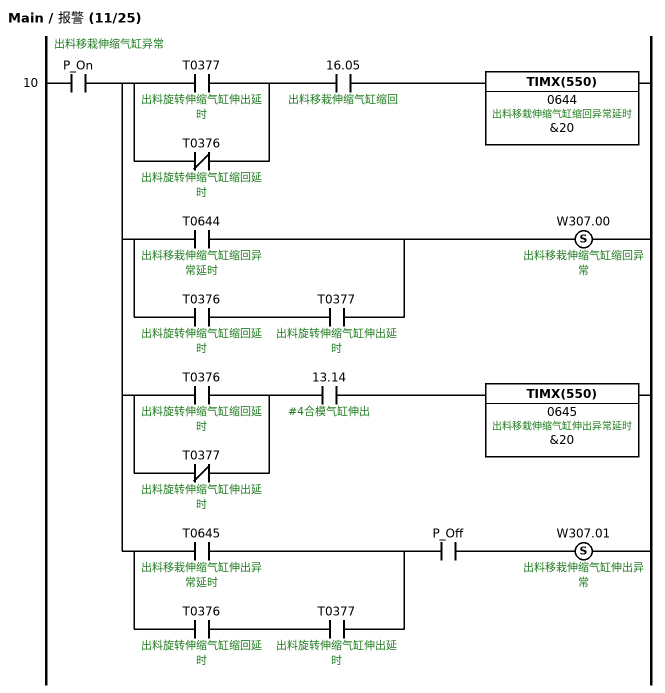
; rung 10: 出料移栽伸缩气缸异常
LD P_On
OUT TR0
LD T0377  ; 出料旋转伸缩气缸伸出延时
ORNOT T0376  ; 出料旋转伸缩气缸缩回延时
ANDLD
AND 16.05  ; 出料移栽伸缩气缸缩回
TIMX(550) 0644 &20  ; 出料移栽伸缩气缸缩回异常延时
LD TR0
LD T0644  ; 出料移栽伸缩气缸缩回异常延时
LD T0376  ; 出料旋转伸缩气缸缩回延时
AND T0377  ; 出料旋转伸缩气缸伸出延时
ORLD
ANDLD
SET W307.00  ; 出料移栽伸缩气缸缩回异常
LD TR0
LD T0376  ; 出料旋转伸缩气缸缩回延时
ORNOT T0377  ; 出料旋转伸缩气缸伸出延时
ANDLD
AND 13.14  ; #4合模气缸伸出
TIMX(550) 0645 &20  ; 出料移栽伸缩气缸伸出异常延时
LD TR0
LD T0645  ; 出料移栽伸缩气缸伸出异常延时
LD T0376  ; 出料旋转伸缩气缸缩回延时
AND T0377  ; 出料旋转伸缩气缸伸出延时
ORLD
ANDLD
AND P_Off
SET W307.01  ; 出料移栽伸缩气缸伸出异常

